{attribute 'qualified_only'}
{attribute 'strict'}
TYPE ST_LaudaReadWriteError :
STRUCT
	SendCommand			: STRING(100);
	ResponseErrorInfo	: E_LaudaResponseError;
END_STRUCT
END_TYPE

(* stored: Version 1.1.0.1, ProductVersion 3.1.4024.13
   DUT ST_LaudaReadWriteError: Id {78ed41a8-ae88-03f3-1bee-690a8c409507} *)
